// TIA Portal V17 export
// export: Created 2026-04-13T11:12:42.3691653Z, ExportSetting WithDefaults, DisplayName Totally Integrated Automation Portal, DisplayVersion V17 Update 4, DisplayName TIA Portal Openness, DisplayVersion V17 Update 4, DisplayName TIA Portal Version Control Interface, DisplayVersion V17, DisplayName SINAMICS Startdrive Advanced, DisplayVersion V17, DisplayName SINAMICS Startdrive G130, G150, S120, S150, SINAMICS MV, S210, DisplayVersion V17, DisplayName SINAMICS Startdrive G110M, G120, G120C, G120D, G120P, G115D, DisplayVersion V17, DisplayName STEP 7 Professional, DisplayVersion V17 Update 4, DisplayName STEP 7 Safety, DisplayVersion V17, DisplayName WinCC Professional, DisplayVersion V17 Update 4
FUNCTION "数组最大平均值" : Void   // FC34, SCL
{ S7_Optimized_Access := 'TRUE' }
VERSION : 0.1
// stored: AutoNumber true, IsIECCheckEnabled false, SetENOAutomatically false, UDAEnableTagReadback false
   VAR_INPUT
      输入数组 : Variant;   // 输入的数组，这里是泛型类型(P#这种数组指针写法)
   END_VAR
   VAR_OUTPUT
      max_out : Variant;   // 最大值输出（无效输出）
      最大值在数组内的索引 : DInt;   // 最大值索引（由于输入数组的类型不确定，无法给出最大值，只能得到数组最大值的索引，其他地方通过索引去访问）
      报错消息 : String;   // 报错消息
      平均值 : LReal;   // 平均值
   END_VAR
   VAR_TEMP
      arr_length : DInt;   // 传入数组的长度值
      i : DInt;   // 循环次数
      arr_int_temp : Array[0..#max_length] of Int;   // 把输入的数组暂存变量int
      max_number_temp_int : Int;   // 最大值暂存int
      arr_real_temp : Array[0..#max_length] of Real;   // 把输入的数组暂存变量real
      max_number_temp_real : Real;   // 最大值的暂存real
      max_index_temp : DInt;   // 最大值的索引暂存
      sum : LReal;   // 数组和
   END_VAR
   VAR CONSTANT
      max_length : DInt := 201;   // 所能处理的最大数组长度，可修改
   END_VAR
BEGIN
   //本程序的数组输入索引是必须从0开始
   IF IS_ARRAY(#输入数组) THEN //判断是否是数组

       #arr_length := UDINT_TO_DINT(CountOfElements(#输入数组)); //找到数组的长度，函数返回值类型是UDINT,要转成DINT

       IF #arr_length < #max_length THEN //如果输入的数组的长度小于设定的最大长度 则进行以下判断

           //**************************判断数组是整数进行计算***************************************

           IF TypeOfElements(#输入数组) = Int THEN //判断输入数组的类型

               VariantGet(SRC := #输入数组,

                          DST => #arr_int_temp);

               #max_number_temp_int := #arr_int_temp[0]; //把索引为0的数认为是最大值

               #max_index_temp := 0; //把0索引存起来

               FOR #i := 0 TO #max_length - 1 DO //循环 从最小索引开始，到最大索引结束

                   IF #max_number_temp_int < #arr_int_temp[#i] THEN //如果最大值小于后面索引的值

                       #max_number_temp_int := #arr_int_temp[#i]; //则把后面索引的值存入最大值变量里

                       #max_index_temp := #i; //再把索引存起来

                   END_IF;

                   #sum := #sum + #arr_int_temp[#i];

               END_FOR;

               VariantPut(SRC := #max_number_temp_int,

                          DST := #max_out); //把最大值输出 int

               #最大值在数组内的索引 := #max_index_temp; //把最大值的索引输出

               #平均值 := #sum / #arr_length;

               //*******************************如果数组是浮点进行计算*********************************

           ELSIF TypeOfElements(#输入数组) = Real THEN //判断输入数组的类型

               VariantGet(SRC := #输入数组,

                          DST => #arr_real_temp); //把输入的数组传入到内部数组进行处理

               #max_number_temp_real := #arr_real_temp[0]; //把索引为0的数认为是最大值

               #max_index_temp := 0; //把0索引存起来

               FOR #i := 0 TO #max_length - 1 DO //循环 从最小索引开始，到最大索引结束

                   IF #max_number_temp_real < #arr_real_temp[#i] THEN //如果最大值小于后面索引的值

                       #max_number_temp_real := #arr_real_temp[#i]; //则把后面索引的值存入最大值变量里

                       #max_index_temp := #i; //再把索引存起来

                   END_IF;

                   #sum := #sum + #arr_real_temp[#i];

               END_FOR;

               VariantPut(SRC := #max_number_temp_real,

                          DST := #max_out); //把最大值输出 real

               #最大值在数组内的索引 := #max_index_temp; //把最大值的索引输出

               #平均值 := #sum / #arr_length;

           END_IF;

       ELSE

           #报错消息 := 'fault'; //如果输入的数组长度超过200个，那就报错

       END_IF;

   END_IF;
END_FUNCTION
